// SIMATIC S7-200 project (STEP 7-Micro/WIN), CPU 224 REL 02.00

ORGANIZATION_BLOCK MAIN:OB1
TITLE=PROGRAM COMMENTS
BEGIN
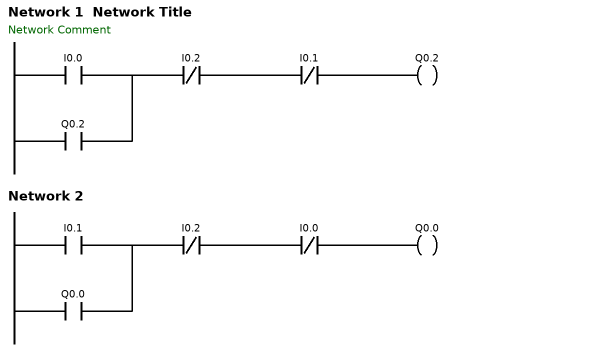
Network 1 // Network Title
// Network Comment
LD     I0.0
O      Q0.2
AN     I0.2
AN     I0.1
=      Q0.2
Network 2
LD     I0.1
O      Q0.0
AN     I0.2
AN     I0.0
=      Q0.0
END_ORGANIZATION_BLOCK
